FUNCTION proj8_TupleStruct_1: REAL
{ S7_Optimized_Access := 'false' }
    VAR_INPUT
        tuple: TupleStruct_1;
    END_VAR

BEGIN
    proj8_TupleStruct_1 := tuple.field8;
END_FUNCTION
